// TIA Portal V17 export
// export: Created 2024-08-09T12:53:14.9915921Z, ExportSetting WithDefaults, DisplayName Totally Integrated Automation Portal, DisplayVersion V17 Update 7, DisplayName TIA Portal Openness, DisplayVersion V17 Update 7, DisplayName TIA Portal Version Control Interface, DisplayVersion V17, DisplayName STEP 7 Professional, DisplayVersion V17 Update 7, DisplayName STEP 7 Safety, DisplayVersion V17 Update 6, DisplayName WinCC Professional, DisplayVersion V17 Update 7
VAR_GLOBAL   // PLC tag table "Dec_Niveaux_Charg"
END_VAR
VAR_GLOBAL CONSTANT   // user constants
   N_DEBLOT : USInt := 1;   // Niveau prise en compte du lot
   N_PRET : USInt := 10;   // Niveau pret
   N_ENCH : USInt := 200;
   N_PP : USInt := 20;   // Niveau presence produit
   N_FINLOT : USInt := 255;   // fin du lot
   NIV_SURPONT_ATT_DEM_CIR : USInt := 10;
   NIV_SURPONT_DEM_CIR : USInt := 20;
   NIV_SURPONT_CHARG_EC : USInt := 40;
   NIV_SURPONT_CONF_FIN_CHAR : USInt := 50;
   NIV_SURPONT_VID_CIR : USInt := 60;
   NIV_SURPONT_FVID_CIR : USInt := 160;
   NIV_SURPONT_ATT_FINLOT : USInt := 200;
   NIV_SURPONT_CIRCUIT_PRET : USInt := 30;
END_VAR
